FUNCTION_BLOCK DataPanel_xDB_08_PVE_SAE_J1939 (* Service Interface Function Block Type *)
  (* Standard: SAE J1939; Function: PVG Valve Driver; Type: DP-34044-7-000; Description: Copyright (c) 2018, 2023 Jose Cabral, HR Agrartechnik GmbH This program and the accompanying materials are made available under the terms of the Eclipse Public License 2.0 which is available at https://www.eclipse.org/legal/epl-2.0/ SPDX-License-Identifier: EPL-2.0 this maps to QX *)
  (* Version 1.0, 2018-12-05, Jose Cabral *)
  (* Version 1.1, 2022-08-04, Franz Höpfinger, HR Agrartechnik GmbH *)
  (* Version 1.2, 2023-01-05, Franz Höpfinger, HR Agrartechnik GmbH *)
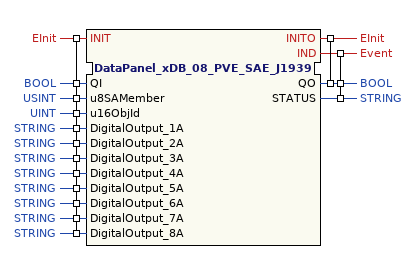
  EVENT_INPUT
    INIT : EInit WITH QI, u8SAMember, u16ObjId, DigitalOutput_1A, DigitalOutput_2A, DigitalOutput_3A, DigitalOutput_4A, DigitalOutput_5A, DigitalOutput_6A, DigitalOutput_7A, DigitalOutput_8A; (* Service Initialization *)
  END_EVENT
  EVENT_OUTPUT
    INITO : EInit WITH QO; (* Initialization Confirm *)
    IND WITH QO, STATUS; (* Indication from Resource *)
  END_EVENT
  VAR_INPUT
    QI : BOOL; (* Event Input Qualifier *)
    u8SAMember : USINT := MI_00; (* Node SA 224..239 *)
    u16ObjId : UINT := ID_NULL; (* Dummy ! set to ID_NULL if in Doubt. ID_OFF deactivates FB. *)
    DigitalOutput_1A : STRING;
    DigitalOutput_2A : STRING;
    DigitalOutput_3A : STRING;
    DigitalOutput_4A : STRING;
    DigitalOutput_5A : STRING;
    DigitalOutput_6A : STRING;
    DigitalOutput_7A : STRING;
    DigitalOutput_8A : STRING;
  END_VAR
  VAR_OUTPUT
    QO : BOOL; (* Event Output Qualifier *)
    STATUS : STRING; (* Service Status *)
  END_VAR
END_FUNCTION_BLOCK
